{attribute addProperty BoxType "KL3356"}
{attribute addProperty Id "Channel_1Channel_5FAA686700"}
{attribute addProperty CRC "2320958694"}
{attribute addProperty SizeInBites "0"}
{attribute addProperty SizeInBytes "0"}
TYPE KL3356_8A5704E6 :
STRUCT
	{attribute addProperty Name "Channel_1"}
	Channel_1 : Channel_5FAA6867;
END_STRUCT
END_TYPE

(* stored: Version 1.2.0.0, ProductVersion 3.1.4024.9
   DUT KL3356_8A5704E6: Id {4a3ba66a-9967-4029-be42-a45c91241e86} *)
